TYPE (* DataPanel Modules with medium IO density DI Struct *)
  (* Version 1.0, 2025-07-21, Franz Höpfinger, initial API and implementation and/or initial documentation *)
  PACKAGE DataPanel::io::MI::DI;
  DataPanel_MI_DI_S : STRUCT
    Pin : USINT := 255;
  END_STRUCT;
END_TYPE
